% RSLogix 500 project Tarea_3_Timers.RSS, saved by version 8.30.00.16 %
PROJECT "UNTITLED"    % processor: MicroLogix 1000 %

PROGRAM FILES
  LAD 2   11 rungs
  LAD 3, 4, 5, 6, 7, 8, 9, 10, 11, 12, 13, 14, 15, 16: only END

DATA FILES
  O0 OUTPUT  1 elements
  I1 INPUT  2 elements
  S2 STATUS  33 elements
  B3 BINARY  32 elements
  T4 TIMER  40 elements
  C5 COUNTER  32 elements
  R6 CONTROL  16 elements
  N7 INTEGER  105 elements

LADDER 2
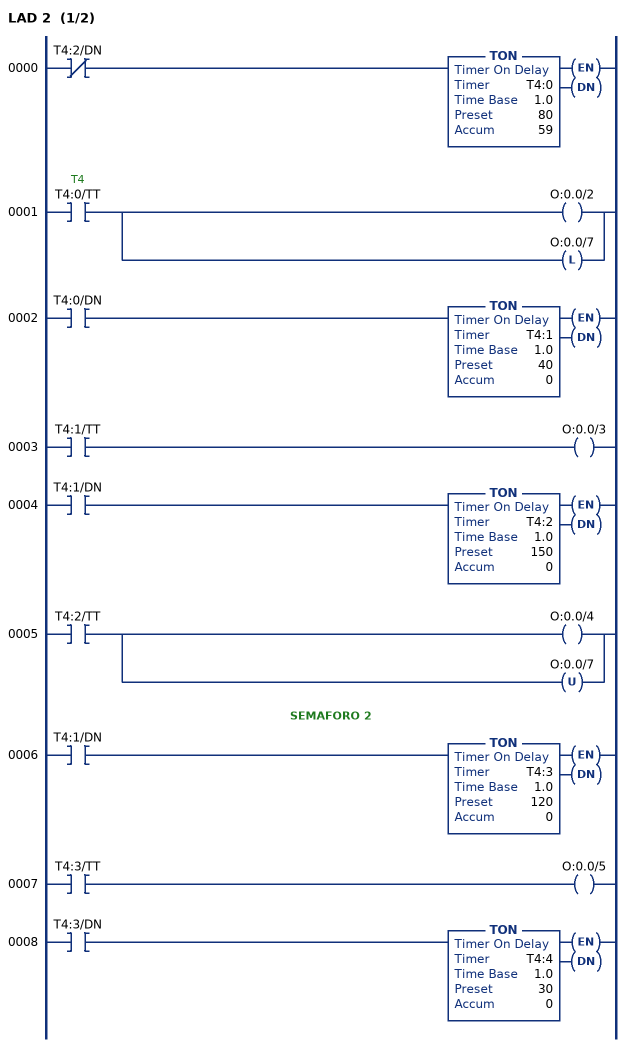
% Rung: 0 %
SOR XIO T4:2/DN TON T4:0 1.0 80 59 EOR
% Rung: 1 %  % edit flag set %
SOR XIC T4:0/TT BST OTE O:0.0/2 NXB OTL O:0.0/7 BND EOR
%   T4:0/TT  T4 %
% Rung: 2 %
SOR XIC T4:0/DN TON T4:1 1.0 40 0 EOR
% Rung: 3 %  % edit flag set %
SOR XIC T4:1/TT OTE O:0.0/3 EOR
% Rung: 4 %
SOR XIC T4:1/DN TON T4:2 1.0 150 0 EOR
% Rung: 5 %  % edit flag set %
SOR XIC T4:2/TT BST OTE O:0.0/4 NXB OTU O:0.0/7 BND EOR
% Rung: 6 %
% TITLE: SEMAFORO 2 %
SOR XIC T4:1/DN TON T4:3 1.0 120 0 EOR
% Rung: 7 %  % edit flag set %
SOR XIC T4:3/TT OTE O:0.0/5 EOR
% Rung: 8 %
SOR XIC T4:3/DN TON T4:4 1.0 30 0 EOR

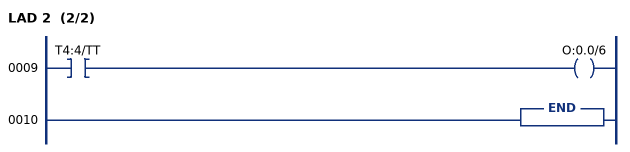
% Rung: 9 %  % edit flag set %
SOR XIC T4:4/TT OTE O:0.0/6 EOR
% Rung: 10 %
SOR END EOR

DATA TABLE (non-zero values as saved)
DATA T4
% .PRE .ACC %
% T4:0 % 80 59
% T4:1 % 40 0
% T4:2 % 150 0
% T4:3 % 120 0
% T4:4 % 30 0
